(* PLC project SafeLOGIC-1, BrAutomation SafeDESIGNER  4.4.0.0 *)
(* stored: companyURL http://www.br-automation.com, creationDateTime Mon Oct 25 15:10:56 2021 *)

PROGRAM Main
  VAR  (* added by the conversion: wires and edge detectors of the diagram *)
    _AND_S58_OUT : ANY;
    _SAFEBOOL_TO_BOOL19_OUT : BOOL;
  END_VAR

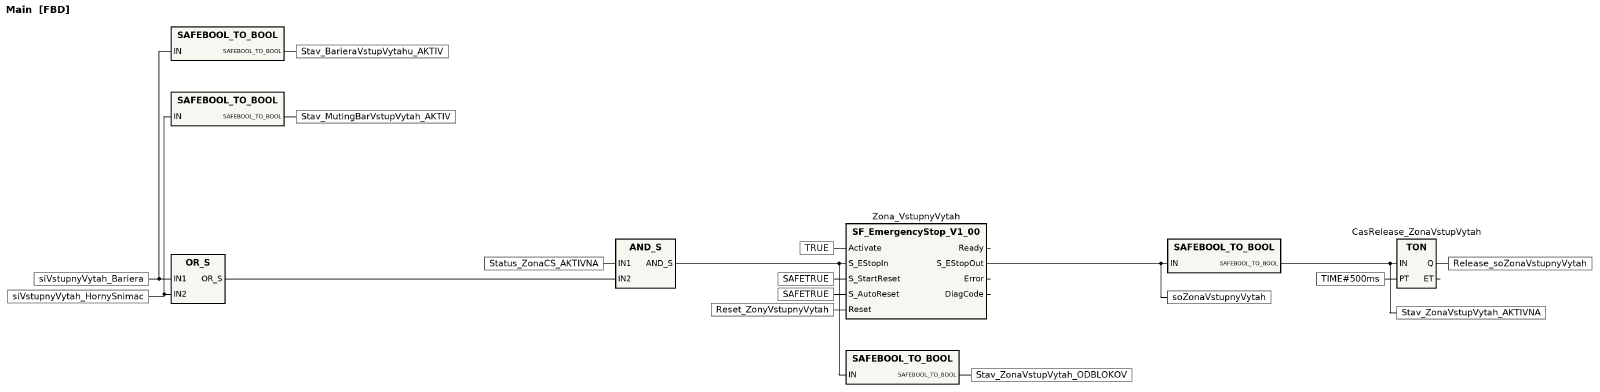
(* FBD diagram, written out as Structured Text *)
_AND_S58_OUT := AND_S(Status_ZonaCS_AKTIVNA, OR_S(siVstupnyVytah_Bariera, siVstupnyVytah_HornySnimac));
Zona_VstupnyVytah(Activate := TRUE, S_EStopIn := _AND_S58_OUT, S_StartReset := SAFETRUE, S_AutoReset := SAFETRUE, Reset := Reset_ZonyVstupnyVytah);
soZonaVstupnyVytah := Zona_VstupnyVytah.S_EStopOut;
_SAFEBOOL_TO_BOOL19_OUT := SAFEBOOL_TO_BOOL(Zona_VstupnyVytah.S_EStopOut);
CasRelease_ZonaVstupVytah(IN := _SAFEBOOL_TO_BOOL19_OUT, PT := TIME#500ms);
Release_soZonaVstupnyVytah := CasRelease_ZonaVstupVytah.Q;
Stav_BarieraVstupVytahu_AKTIV := SAFEBOOL_TO_BOOL(siVstupnyVytah_Bariera);
Stav_ZonaVstupVytah_ODBLOKOV := SAFEBOOL_TO_BOOL(_AND_S58_OUT);
Stav_ZonaVstupVytah_AKTIVNA := _SAFEBOOL_TO_BOOL19_OUT;
Stav_MutingBarVstupVytah_AKTIV := SAFEBOOL_TO_BOOL(siVstupnyVytah_HornySnimac);
END_PROGRAM
